// Mitsubishi GX Works2 project: 231003-001- exercicios-1   PLC: Q03UDV

// global labels: Global1
VAR_GLOBAL
  Up_Down AT M34 : BOOL;
END_VAR

// task Task_01 (event TRUE, interval 0, priority 31): POU_01

PROGRAM POU_01
VAR
  CTD_1 : CTD;
  CTU_1 : CTU;
  meuc : CTU;
  novo : CTUD;
  TP_1 : TP;
  TON_1 : TON;
  TOF_1 : TOF;
  dr : TIME;
  timetp : TIME;
  timeon : TIME;
  TimeOFF : TIME;
  Input : BOOL;
  red : BOOL;
  TP_2 : TP;
  ver : BOOL;
  verd : BOOL;
  TP_3 : TP;
  amar : BOOL;
END_VAR
(* structured ladder/FBD written out as ST: instructions are called as NAME(EN, inputs, outputs); _pN, _eN, _tN stand for wires *)
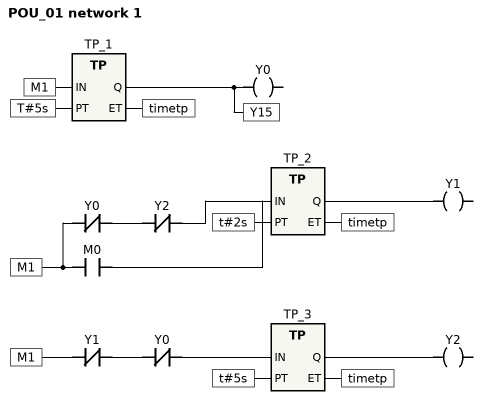
(* network 1 *)
TP_1(IN := M1, PT := T#5s, ET => timetp);
Y15 := TP_1.Q;
Y0 := TP_1.Q;
TP_2(IN := (M1 AND NOT Y0 AND NOT Y2) OR (M1 AND M0), PT := t#2s, ET => timetp);
Y1 := TP_2.Q;
TP_3(IN := M1 AND NOT Y1 AND NOT Y0, PT := t#5s, ET => timetp);
Y2 := TP_3.Q;
END_PROGRAM
